FUNCTION_BLOCK AX_FB_RS_T_FF (* Realizes a bistable reset-dominat latch plus Toggle (with Adapter) *)
  (* Standard: 61499-1; Description: Copyright (c) 2023 Martin Erich Jobst, HR Agrartechnik GmbH This program and the accompanying materials are made available under the terms of the Eclipse Public License 2.0 which is available at https://www.eclipse.org/legal/epl-2.0/ SPDX-License-Identifier: EPL-2.0 *)
  (* Version 3.0, 2025-04-14, Patrick Aigner, changed package *)
  (* Version 1.0, 2023-04-28, Martin Jobst, initial API and implementation and/or initial documentation *)
  PACKAGE adapter::bistableElements;
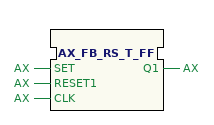
  SOCKETS
    SET : adapter::types::unidirectional::AX; (* Set *)
    RESET1 : adapter::types::unidirectional::AX; (* Reset *)
    CLK : adapter::types::unidirectional::AX; (* Clock *)
  END_SOCKETS
  PLUGS
    Q1 : adapter::types::unidirectional::AX; (* Output *)
  END_PLUGS
  VAR
    EDGE : BOOL := FALSE;
  END_VAR
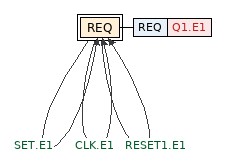
  EC_STATES
    REQ : REQ -> Q1.E1;
  END_STATES
  EC_TRANSITIONS
    REQ TO REQ := RESET1.E1;
    REQ TO REQ := SET.E1;
    REQ TO REQ := CLK.E1;
  END_TRANSITIONS
  ALGORITHM REQ IN ST:
IF RESET1.D1 THEN
	Q1.D1 := BOOL#FALSE;
ELSIF SET.D1 THEN
	Q1.D1 := BOOL#TRUE;
ELSIF CLK.D1 AND NOT EDGE THEN
	Q1.D1 := NOT Q1.D1;
END_IF;
EDGE := CLK.D1;
  END_ALGORITHM
END_FUNCTION_BLOCK
